{attribute addProperty BoxType "EL1512-0000-0016"}
{attribute addProperty Id "Set_counterAT %Q*BOOL813Inhibit_counterAT %Q*BOOL814Set_counter_valueAT %Q*UDINT32417"}
{attribute addProperty CRC "4004019521"}
{attribute addProperty SizeInBites "48"}
{attribute addProperty SizeInBytes "6"}
TYPE CNT_Outputs_Channel_EEA87D41 :
STRUCT
	{attribute addProperty Name "Set_counter"}
	Set_counter AT %Q* : BOOL;
	{attribute addProperty Name "Inhibit_counter"}
	Inhibit_counter AT %Q* : BOOL;
	{attribute addProperty Name "Set_counter_value"}
	Set_counter_value AT %Q* : UDINT;
END_STRUCT
END_TYPE

(* stored: Version 1.2.0.0, ProductVersion 3.1.4024.9
   DUT CNT_Outputs_Channel_EEA87D41: Id {37767990-a36b-4a39-99fc-f3bf6e392c7e} *)
